FUNCTION F_REAL_ARG : ST_Arg
VAR_INPUT
	fInput : REAL;
END_VAR
VAR
	stArg : ST_Arg;
	sysVar_Info : __SYSTEM.VAR_INFO;
END_VAR

sysVar_Info 	:= __VARINFO(fInput);
stArg.TypeClass := sysVar_Info.TypeClass;
stArg.pValue 	:= 0;
stArg.diSize 	:= SIZEOF(fInput);
stArg.sValue 	:= TO_STRING(fInput); 
F_REAL_ARG := stArg;

END_FUNCTION

(* stored: Version 1.1.0.1, ProductVersion 3.1.4024.4
   POU F_REAL_ARG: Id {ba8eba09-8499-4b1e-b280-e114003bc388}, SpecialFunc None *)
